FUNCTION_BLOCK fb_maptest (* Minimal FB for mapping tests *)
  (* Standard: 61499-1 *)
  (* Version 1.0, 2026-02-23, test, 4diac tests *)
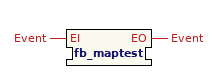
  EVENT_INPUT
    EI;
  END_EVENT
  EVENT_OUTPUT
    EO;
  END_EVENT
  EC_STATES
    START; (* Initial State *)
  END_STATES
END_FUNCTION_BLOCK
